# EPICS substitutions: public/db/user.substitutions
# Example substitutions file

file "db/circle.db" {
    { user = "may" }
}

file "db/dbExample1.db" {
    { user = "may" }
}

file "db/bangs.db" {
    pattern { user, no, scan, initValue, expression }
        { "may", 1, "1 second", "1.23274", "(A<=B && A>=D)?A+cos(C*PI/180):D" }
        { "may", 2, "6 second", "0.99875", "(A<=B && A>=D)?A+tan(C*PI/180-PI/2):D" }
        { "may", 3, "9 second", "1.16729", "(A<=B && A>=D)?A+cos(C*PI/180):D" }
        { "may", 4, "3 second", "1.23274", "(A<=B && A>=D)?A+cos(C*PI/180):D" }
        { "may", 5, "7 second", "1.19371", "(A<=B && A>=D)?A+tan(C*PI/180-PI/2):D" }
        { "may", 6, "5 second", "1.11274", "(A<=B && A>=D)?A+cos(C*PI/180):D" }
        { "may", 7, "1 second", "1.03671", "(A<=B && A>=D)?A+cos(C*PI/180):D" }
        { "may", 8, "10 second", "1.39877", "(A<=B && A>=D)?A+tan(C*PI/180-PI/2):D" }
        { "may", 9, "5 second", "1.96729", "(A<=B && A>=D)?A+cos(C*PI/180):D" }
        { "may", 10, "10 second", "1.03274", "(A<=B && A>=D)?A+cos(C*PI/180):D" }
        { "may", 11, "4 second", "1.04172", "(A<=B && A>=D)?A+tan(C*PI/180-PI/2):D" }
        { "may", 12, ".5 second", "1.19739", "(A<=B && A>=D)?A+cos(C*PI/180):D" }
        { "may", 13, "3 second", "1.02417", "(A<=B && A>=D)?A+cos(C*PI/180):D" }
        { "may", 14, "9 second", "1.19198", "(A<=B && A>=D)?A+tan(C*PI/180-PI/2):D" }
        { "may", 15, "5 second", "1.13167", "(A<=B && A>=D)?A+cos(C*PI/180):D" }
        { "may", 16, "10 second", "1.20271", "(A<=B && A>=D)?A+cos(C*PI/180):D" }
        { "may", 17, "2 second", "1.30173", "(A<=B && A>=D)?A+tan(C*PI/180-PI/2):D" }
        { "may", 18, "5 second", "1.29712", "(A<=B && A>=D)?A+cos(C*PI/180):D" }
        { "may", 19, "3 second", "1.12421", "(A<=B && A>=D)?A+cos(C*PI/180):D" }
}
file "db/bars.db" {
    pattern { user, no, scan, initValue, expression }
        { "may", 1, "1 second", "611.124359", "(A<=B && A>=D)?A+cos(C*PI/180)*31.177:D" }
        { "may", 2, "3 second", "598.83727", "(A<=B && A>=D)?A+cos(C*PI/180)*29.73:D" }
        { "may", 3, "4 second", "572.91024", "(A<=B && A>=D)?A+cos(C*PI/180)*31.177:D" }
        { "may", 4, "3 second", "601.07129", "(A<=B && A>=D)?A+cos(C*PI/180)*31.177:D" }
        { "may", 5, "7 second", "549.12943", "(A<=B && A>=D)?A+cos(C*PI/180)*29.73:D" }
        { "may", 6, "5 second", "558.23951", "(A<=B && A>=D)?A+cos(C*PI/180)*31.177:D" }
        { "may", 7, "1 second", "592.12351", "(A<=B && A>=D)?A+cos(C*PI/180)*31.177:D" }
        { "may", 8, "10 second", "587.34826", "(A<=B && A>=D)?A+cos(C*PI/180)*31.177:D" }
        { "may", 9, "2 second", "593.00281", "(A<=B && A>=D)?A+cos(C*PI/180)*31.177:D" }
        { "may", 10, ".5 second", "621.11729", "(A<=B && A>=D)?A+cos(C*PI/180)*31.177:D" }
}

file db/dbExample2.db {
    pattern { user, no, scan }
        { "may", 1, "1 second" }
        { "may", 2, "2 second" }
        { "may", 3, "5 second" }
}

file "db/tankBars.db" {
    { user = "may" }
}

file "db/leds.db" {
    pattern { user, no, scan }
        { "may", 0, "1 second" }
        { "may", 1, "3 second" }
        { "may", 2, "5 second" }
        { "may", 3, "2 second" }
}
